PROGRAM prgComEffIO
VAR
	fbCom		: FB_MqttCommunicator_V2;
END_VAR

fbCom(
	bConnect:= TRUE, 
	strAuthKey:= 'BE736352867778' , 
	sUserName:= '357937e6-a18b-481e-8d82-4d957ba896c8', 
	sUserPassword:= 'eb079f87-6065-4dfe-8b33-960e910d1962' , 
	eSavePositionCertificate:= eSavePositionOnPLC.ePostionHardDisk , 
	time_HeartBeat_sec:= , 
	bConnected=> , 
	bError=> , 
	hrErrorCode=> , 
	eConnectionState=> , 
	eErrorMessage_Out=> );

(* old
fbCom(
	bConnect:= TRUE, 
	sUserName:= '4bd5671c-5161-4477-be33-80f6ab0ab0ea', 
	sUserPassword:= 'a9f16306-5d85-4294-8f17-fbe4adf6f24f', 
	eSavePositionCertificate:= eSavePositionOnPLC.ePostionHardDisk, 
	bConnected=> , 
	bError=> , 
	hrErrorCode=> , 
	eConnectionState=> , 
	eErrorMessage_Out=> );
*)

END_PROGRAM

(* stored: Version 1.1.0.1, ProductVersion 3.1.4024.11
   POU prgComEffIO: Id {cbcd318b-bf51-484c-bcaa-d6efcdf43fe3}, SpecialFunc None *)
